TYPE ST_ITC_FunctionEmulation :
(**************************************************************************************
 * 	Application		:	BoxControl Framework
 *	Revision		:	$Revision: 404529 $
 *	Revision date	:	$Date: 2018-04-23 08:21:38 +0200 (Mo., 23 Apr 2018) $
 *	Last changed by	:	$Author: b7bolm $
 *	URL				:	$URL: http://almscdc.swisslog.com/repo/SWPD/Development/BoxControlFramework/20_Release/trunk/01_Software/BCF/BCF/JumpStart/20_Product/11_Emu/12_E_Functions/10_Lib/10_Conv/01_DUTs/ST_ITC_FunctionEmulation.TcDUT $
 *
 *	Purpose			:	Function ITC structures
 *
 * ------------------------------------------------------------------------------------
 *	Copyright Swisslog [IP AG], Switzerland. All rights reserved.
 * 
 * ------------------------------------------------------------------------------------
 *	
 * 	Revision History: 
 *
 * 	VERSION			DATE			INITIALS			DESCRIPTION
 *	0.1				01.01.2001		swl					Example
 *
 **************************************************************************************)
STRUCT
	FunctionITC	: ST_ITC_FunctionITC_Emulation; // ITC function data
	ZoneITC		: ARRAY [1..NUMBER_OF_ZONES_PER_FUNCTION] OF ST_ITC_ZoneEmulation; // ITC Zone data	
END_STRUCT
END_TYPE

(* stored: Version 1.1.0.1, ProductVersion 3.1.4022.12
   DUT ST_ITC_FunctionEmulation: Id {4f5af6e2-5cb8-4562-8a98-709ade4b7320} *)
